// TIA Portal V15.1 export
// export: Created 2024-06-21T08:41:09.0371429Z, ExportSetting WithDefaults, DisplayName Totally Integrated Automation Portal, DisplayVersion V15.1 Update 5, DisplayName TIA Portal Openness, DisplayVersion V15.1 Update 5, DisplayName SINAMICS Startdrive Advanced, DisplayVersion V15.1, DisplayName G130, G150, S120, S150, SINAMICS MV, S210, DisplayVersion V15.1, DisplayName G110M, G120, G120C, G120D, G120P, DisplayVersion V15.1, DisplayName STEP 7 Professional, DisplayVersion V15.1 Update 5, DisplayName STEP 7 Safety, DisplayVersion V15.1, DisplayName WinCC Professional, DisplayVersion V15.1 Update 5, DisplayName SIMATIC Visualization Architect, DisplayVersion V15.1
FUNCTION "LGBProcessLighting-Config" : Void   // FC6697, FBD
TITLE = LGBProcessLighting-Config
{ S7_Optimized_Access := 'TRUE' }
VERSION : 0.1
// stored: AutoNumber false, IsIECCheckEnabled false, SetENOAutomatically False, UDAEnableTagReadback false
   VAR_INPUT
      C_WorkStationNr : Int;   // Workstation number
      C_MaxWorkStations : Int;   // Maximum of workstation
      C_Intensity1Used : Bool;   // Intensity1 is used
      C_ColourGroupIntensity1 : Int;   // Colour group for Intensity 1
      C_ColourGroupIntensity1Desc : String;   // Description Colour group for Intensity 1
      C_Intensity2Used : Bool;   // Intensity2 is used
      C_ColourGroupIntensity2 : Int;   // Colour group for Intensity 2
      C_ColourGroupIntensity2Desc : String;   // Description Colour group for Intensity 2
      C_Intensity3Used : Bool;   // Intensity3 is used
      C_ColourGroupIntensity3 : Int;   // Colour group for Intensity 3
      C_ColourGroupIntensity3Desc : String;   // Description Colour group for Intensity 3
      C_DelayBreakMode : Time;   // Delay time for create Breake mode is the production line is stopped
   END_VAR
   VAR_IN_OUT
      IO_Config : "ProcessLightingConfig";   // Config
   END_VAR
BEGIN

REGION Network 1: **** 8 - Outputs **** Move Config
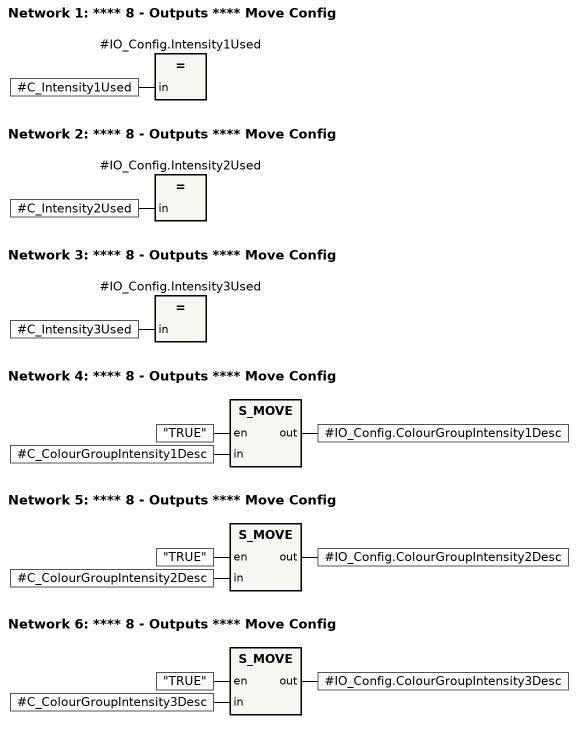
   #IO_Config.Intensity1Used := #C_Intensity1Used;
END_REGION

REGION Network 2: **** 8 - Outputs **** Move Config
   #IO_Config.Intensity2Used := #C_Intensity2Used;
END_REGION

REGION Network 3: **** 8 - Outputs **** Move Config
   #IO_Config.Intensity3Used := #C_Intensity3Used;
END_REGION

REGION Network 4: **** 8 - Outputs **** Move Config
   IF "TRUE" THEN #IO_Config.ColourGroupIntensity1Desc := #C_ColourGroupIntensity1Desc; END_IF;
END_REGION

REGION Network 5: **** 8 - Outputs **** Move Config
   IF "TRUE" THEN #IO_Config.ColourGroupIntensity2Desc := #C_ColourGroupIntensity2Desc; END_IF;
END_REGION

REGION Network 6: **** 8 - Outputs **** Move Config
   IF "TRUE" THEN #IO_Config.ColourGroupIntensity3Desc := #C_ColourGroupIntensity3Desc; END_IF;
END_REGION

NETWORK
TITLE = **** 8 - Outputs **** Move Config UDT
// Move Config
      L     #C_WorkStationNr;
      T     #IO_Config.WorkStationNr;
      L     #C_MaxWorkStations;
      T     #IO_Config.MaxWorkStations;
      L     #C_ColourGroupIntensity1;
      T     #IO_Config.ColourGroupIntensity1;
      L     #C_ColourGroupIntensity2;
      T     #IO_Config.ColourGroupIntensity2;
      L     #C_ColourGroupIntensity3;
      T     #IO_Config.ColourGroupIntensity3;
      L     #C_DelayBreakMode;
      T     #IO_Config.DelayBreakMode;
END_FUNCTION
